TYPE ST_TwoHandParCfg :
STRUCT
    SchemaVersion : UINT := 1;
    RequireReleaseBetweenCycles : BOOL := TRUE;
END_STRUCT
END_TYPE

(* stored: Version 1.1.0.1, ProductVersion 3.1.4024.12
   DUT ST_TwoHandParCfg: Id {813a0d49-41a5-4db1-b348-08d26f2cce75} *)
